(* IEC 61131-3 sources: paho.mqtt.c-ar/Samples/IotMqttSamples/SampleTasks/WebSocketSSL, 2 files *)

(* ---- Main.st ---- *)
PROGRAM _CYCLIC

	Parameters;

	IotMqttClient_0.Enable			:= TRUE;
	IotMqttClient_0.Connect			:= TRUE;
	IotMqttClient_0.IotMqttLink 	:= ADR(IotMqttLink);
	IotMqttClient_0.Parameters		:= IotMqttParameters;
	IotMqttClient_0();

	PublishTopic	:= 'B&R_DemoProject/WSS';
	brsstrcat(ADR(PublishTopic),ADR(ClientID));

	Subscribe;
	Publish;
END_PROGRAM

PROGRAM _EXIT

    IotMqttClient_0(Enable	:= FALSE);
    IotMqttPublish_0(Enable	:= FALSE);
    IotMqttSubscribe_0(Enable := FALSE);

END_PROGRAM

(* ---- Parameters.st ---- *)
ACTION Parameters:

	//Prepare Client ID. Add a timestamp to ensure any client will repeat it
	UtcDTGetTime_0(enable := TRUE);
	IF brsstrcmp(ADR(ClientID),ADR('')) = 0 THEN
		ClientID := 'B&R_Demo_';
		ST_name(0,ADR(ThreadName),0);
		brsstrcat(ADR(ClientID),ADR(ThreadName));
		brsstrcat(ADR(ClientID),ADR("_"));
		brsmemset(ADR(AuxString),0,SIZEOF(AuxString));
		AuxString := UDINT_TO_STRING(DT_TO_UDINT(UtcDTGetTime_0.DT1));
		brsstrcat(ADR(ClientID),ADR(AuxString));	//Timestamp
	END_IF

	IotMqttParameters.ServerUri				:= 'test.mosquitto.org';
	IotMqttParameters.ConnectionType		:= IotMqtt_WS;	//Use websocket with tls
	IotMqttParameters.Port					:= 8081;
	IotMqttParameters.TLS.UseTLS			:= TRUE;
	IotMqttParameters.ClientID				:= ClientID;
	IotMqttParameters.CleanSession			:= TRUE;
	IotMqttParameters.KeepAliveInterval		:= T#20s;
	IotMqttParameters.AutomaticReconnect	:= TRUE;

END_ACTION
